FUNCTION_BLOCK ATM_SPLIT_SIGNED (* Teilt einen TIME-Wert in 2 einseitige Betragswerte auf (z.B. fuer 2 getrennte Bargraphen links/rechts einer Mittelstellung): NEG_MAG = MAX(0,-Y), POS_MAG = MAX(0,Y). Jede Seite feuert ihr Event nur bei tatsaechlicher Wertaenderung gegenueber ihrem eigenen aktuellen Ausgangswert (nicht bei jedem Y-Update), analog zu AX_OR_2 ("Adapter-Ausgang wird nur bei Wertaenderung aktualisiert") - wichtig, wenn Y lange auf einer Seite bleibt und die andere Seite konstant 0 haelt. *)
  (* Standard: 61499-2 *)
  (* Version 2.1, 2026-09-11, Franz Höpfinger, Kein eigener prevNeg/prevPos-Internal mehr noetig - Vergleich direkt gegen NEG_MAG.D1/POS_MAG.D1 (Plug-Ausgang haelt den letzten Wert bereits selbst) *)
  (* Version 2.0, 2026-09-11, Franz Höpfinger, Event nur noch bei tatsaechlicher Wertaenderung je Seite (vorher: bei jedem Y-Update immer beide Events, unabhaengig ob sich der Wert aendert) *)
  (* Version 1.0, 2026-09-11, Franz Höpfinger, Typfamilie zu AR_SPLIT_SIGNED, generisch fuer jede aehnliche Anzeige *)
  PACKAGE adapter::Engineering::splitting::signed;
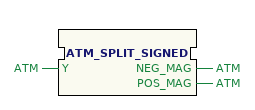
  SOCKETS
    Y : adapter::types::unidirectional::ATM; (* Eingangswert *)
  END_SOCKETS
  PLUGS
    NEG_MAG : adapter::types::unidirectional::ATM; (* MAX(0, -Y) - Betrag der negativen Auslenkung, Event nur bei Aenderung *)
    POS_MAG : adapter::types::unidirectional::ATM; (* MAX(0, Y) - Betrag der positiven Auslenkung, Event nur bei Aenderung *)
  END_PLUGS
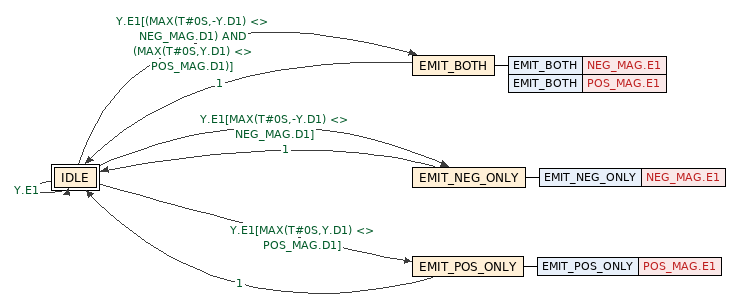
  EC_STATES
    IDLE; (* Initial State *)
    EMIT_BOTH : EMIT_BOTH -> NEG_MAG.E1, EMIT_BOTH -> POS_MAG.E1;
    EMIT_NEG_ONLY : EMIT_NEG_ONLY -> NEG_MAG.E1;
    EMIT_POS_ONLY : EMIT_POS_ONLY -> POS_MAG.E1;
  END_STATES
  EC_TRANSITIONS
    IDLE TO EMIT_BOTH := Y.E1[(MAX(T#0S,-Y.D1) <> NEG_MAG.D1) AND (MAX(T#0S,Y.D1) <> POS_MAG.D1)];
    IDLE TO EMIT_NEG_ONLY := Y.E1[MAX(T#0S,-Y.D1) <> NEG_MAG.D1];
    IDLE TO EMIT_POS_ONLY := Y.E1[MAX(T#0S,Y.D1) <> POS_MAG.D1];
    IDLE TO IDLE := Y.E1;
    EMIT_BOTH TO IDLE := 1;
    EMIT_NEG_ONLY TO IDLE := 1;
    EMIT_POS_ONLY TO IDLE := 1;
  END_TRANSITIONS
  ALGORITHM EMIT_BOTH IN ST:
NEG_MAG.D1 := MAX(T#0S,-Y.D1);
POS_MAG.D1 := MAX(T#0S,Y.D1);
  END_ALGORITHM
  ALGORITHM EMIT_NEG_ONLY IN ST:
NEG_MAG.D1 := MAX(T#0S,-Y.D1);
  END_ALGORITHM
  ALGORITHM EMIT_POS_ONLY IN ST:
POS_MAG.D1 := MAX(T#0S,Y.D1);
  END_ALGORITHM
END_FUNCTION_BLOCK
